{attribute 'GeneratedUsingTerminal: EK1100-0000-0018'}
{attribute addProperty BoxType "EK1100-0000-0018"}
{attribute addProperty Id "Beckhoff_EP4xxxEK1122Beckhoff_EP4xxxEK1122_BC01358E256"}
{attribute addProperty CRC "3148249264"}
{attribute addProperty Size "256"}
TYPE Beckhoff_EP4xxx_BBA678B0 EXTENDS EK1100_1FC0878B :
STRUCT
	{attribute addProperty Name "Beckhoff_EP4xxxEK1122"}
	{attribute addProperty PreviousPort "Beckhoff EP4xxx : B"}
	Beckhoff_EP4xxxEK1122 : Beckhoff_EP4xxxEK1122_BC01358E;
END_STRUCT
END_TYPE

(* stored: Version 1.2.0.0, ProductVersion 3.1.4024.9
   DUT Beckhoff_EP4xxx_BBA678B0: Id {c30ebae8-64e9-46c2-8f27-5674152237db} *)
